FUNCTION F_DWORD2CMYK : ST_ColorCMYK
VAR_INPUT
	Color					: DWORD;
END_VAR

VAR
	stColor					: ST_COLOR;
	tmpArray				: ARRAY[0..3] OF BYTE;
	
	Rc						: REAL;
	Gc						: REAL;
	Bc						: REAL;

	K						: REAL;
	
END_VAR

stColor := F_DWORD2RGB(Color);

Rc := stColor.nRed / 255;
Gc := stColor.nGreen / 255;
Bc := stColor.nBlue / 255;

IF (Rc + Gc + Bc) = 0 THEN
	F_DWORD2CMYK.nCyan := 0;
	F_DWORD2CMYK.nMagenta := 0;
	F_DWORD2CMYK.nYellow := 0;
	F_DWORD2CMYK.nKey := 100;	
	RETURN;
END_IF

K := TO_BYTE(1 - MAX(Rc, MAX(Gc, Bc)));

F_DWORD2CMYK.nCyan := TO_BYTE((1-Rc-K)/(1-K));
F_DWORD2CMYK.nMagenta := TO_BYTE((1-Gc-K)/(1-K));
F_DWORD2CMYK.nYellow := TO_BYTE((1-Bc-K)/(1-K));
F_DWORD2CMYK.nKey := TO_BYTE(K);

END_FUNCTION

(* stored: Version 1.1.0.1
   POU F_DWORD2CMYK: Id {54f5964d-ec4b-4e45-87ee-1cae1b847cb5}, SpecialFunc None *)
